ABB RAPID module: 002FC75C

MODULE CalibData
	CONST robtarget pHome:=[[506.291650772,0,679.49999918],[0.499999994,0,0.866025407,0],[0,0,0,0],[9E+09,9E+09,9E+09,9E+09,9E+09,9E+09]];
	CONST robtarget conveyor:=[[-9.861164677,-596.337827708,208.8592172],[0.048273193,0.711237174,0.699573246,-0.049078048],[-2,-1,0,0],[9E+09,9E+09,9E+09,9E+09,9E+09,9E+09]];
	CONST robtarget Oven:=[[676.77830567,0,798.153707831],[0.500000149,0,0.866025318,0],[0,0,0,0],[9E+09,9E+09,9E+09,9E+09,9E+09,9E+09]];
	CONST robtarget manipulation:=[[40.184227668,785.23645067,592.1503114],[0.554573369,-0.481039839,0.478798532,0.481457181],[0,0,-1,1],[9E+09,9E+09,9E+09,9E+09,9E+09,9E+09]];
ENDMODULE
